FUNCTION POU : BOOL
VAR_INPUT
END_VAR
VAR
END_VAR

END_FUNCTION

(* stored: Version 1.1.0.1, ProductVersion 3.1.4024.10
   POU POU: Id {f05d997b-04f7-443c-bc9a-8b59643a234f}, SpecialFunc None *)
